// TIA Portal project "Module1.2" (V16)

(* hardware
DEVICE "S7-1200 station_1"  S7-1200 Station
   slot 0: "Rack_0"  S7-1200 Rack  Rack  V1.0
   slot 1: "PLC_1"  CPU 1214C DC/DC/DC  6ES7 214-1AG40-0XB0  V4.2
   slot 2: "DI 8/DQ 8x24VDC_1"  SM 1223 DI8/DQ8 x 24VDC  6ES7 223-1BH30-0XB0  V1.0
*)

// ===== PLC "PLC_1"  CPU 1214C DC/DC/DC =====

VAR_GLOBAL   // PLC tag table "Default tag table"
   "R" AT %Q2.1 : Bool;
   "embryoQuality" AT %M10.0 : Bool;
   "initialStep" AT %M0.0 : Bool;
   "reset" AT %M0.1 : Bool;
   "start" AT %M0.2 : Bool;
   "startConveyor" AT %M0.3 : Bool;
   "pushEmbryo" AT %M0.4 : Bool;
   "waitEmbryo" AT %M0.5 : Bool;
   "stopConveyor" AT %M0.6 : Bool;
   "grapEmbryo" AT %M0.7 : Bool;
   "goingUp" AT %M1.0 : Bool;
   "goingDown" AT %M1.1 : Bool;
   "goingRight" AT %M1.2 : Bool;
   "putEmbryoDown" AT %M1.3 : Bool;
   "checkEmbryo" AT %M1.4 : Bool;
   "realizeEmbryo" AT %M1.5 : Bool;
   "offSuction" AT %M1.6 : Bool;
   "fs" AT %I1.0 : Bool;
END_VAR

VAR_GLOBAL   // PLC tag table "Default tag table_1"
   "System_Byte" AT %MB100 : Byte;
   "FirstScan" AT %M100.0 : Bool;
   "DiagStatusUpdate" AT %M100.1 : Bool;
   "AlwaysTRUE" AT %M100.2 : Bool;
   "AlwaysFALSE" AT %M100.3 : Bool;
   "Clock_Byte" AT %MB200 : Byte;
   "Clock_10Hz" AT %M200.0 : Bool;
   "Clock_5Hz" AT %M200.1 : Bool;
   "Clock_2.5Hz" AT %M200.2 : Bool;
   "Clock_2Hz" AT %M200.3 : Bool;
   "Clock_1.25Hz" AT %M200.4 : Bool;
   "Clock_1Hz" AT %M200.5 : Bool;
   "Clock_0.625Hz" AT %M200.6 : Bool;
   "Clock_0.5Hz" AT %M200.7 : Bool;
   "startBTN" AT %I0.0 : Bool;
   "stopBTN" AT %I0.1 : Bool;
   "resetBTN" AT %I0.2 : Bool;
   "headConveyorSS" AT %I0.3 : Bool;
   "enConveyorSS" AT %I0.6 : Bool;
   "embryoSS" AT %I2.1 : Bool;
   "pushCompressLimit" AT %I0.7 : Bool;
   "pushExpandLimit" AT %I2.0 : Bool;
   "leftLimit" AT %I2.6 : Bool;
   "rightLimit" AT %I2.4 : Bool;
   "downLimit" AT %I2.2 : Bool;
   "upLimit" AT %I2.3 : Bool;
   "stopperCompressLimit" AT %I0.4 : Bool;
   "stopperExpandLimit" AT %I0.5 : Bool;
   "middleHCylinder" AT %I2.5 : Bool;
   "Push" AT %Q0.5 : Bool;
   "Left" AT %Q1.1 : Bool;
   "Right" AT %Q0.2 : Bool;
   "Down" AT %Q0.3 : Bool;
   "stopperDown" AT %Q0.0 : Bool;
   "Conveyor" AT %Q2.0 : Bool;
   "Suction" AT %Q0.4 : Bool;
   "Y" AT %Q2.3 : Bool;
   "G" AT %Q2.2 : Bool;
   "CBPL" AT %I2.7 : Bool;
END_VAR

// folder: System blocks/Program resources

DATA_BLOCK "timer1"   // DB1
{ S7_Optimized_Access := 'TRUE' }
AUTHOR : Simatic
FAMILY : IEC
NAME : IEC_TMR
VERSION : 1.0
// stored: InstanceOfName IEC_TIMER
"IEC_TIMER"
BEGIN
END_DATA_BLOCK

DATA_BLOCK "timer2"   // DB2
{ S7_Optimized_Access := 'TRUE' }
AUTHOR : Simatic
FAMILY : IEC
NAME : IEC_TMR
VERSION : 1.0
// stored: InstanceOfName IEC_TIMER
"IEC_TIMER"
BEGIN
END_DATA_BLOCK

DATA_BLOCK "timer3"   // DB3
{ S7_Optimized_Access := 'TRUE' }
AUTHOR : Simatic
FAMILY : IEC
NAME : IEC_TMR
VERSION : 1.0
// stored: InstanceOfName IEC_TIMER
"IEC_TIMER"
BEGIN
END_DATA_BLOCK

// folder: (top level)

ORGANIZATION_BLOCK "Main"   // OB1, LAD, ProgramCycle
TITLE = "Main Program Sweep (Cycle)"
{ S7_Optimized_Access := 'TRUE' }
VERSION : 0.1
   VAR_INPUT
      Initial_Call : Bool;   // Initial call of this OB
      Remanence : Bool;   // =True, if remanent data are available
   END_VAR
BEGIN

REGION Network 1
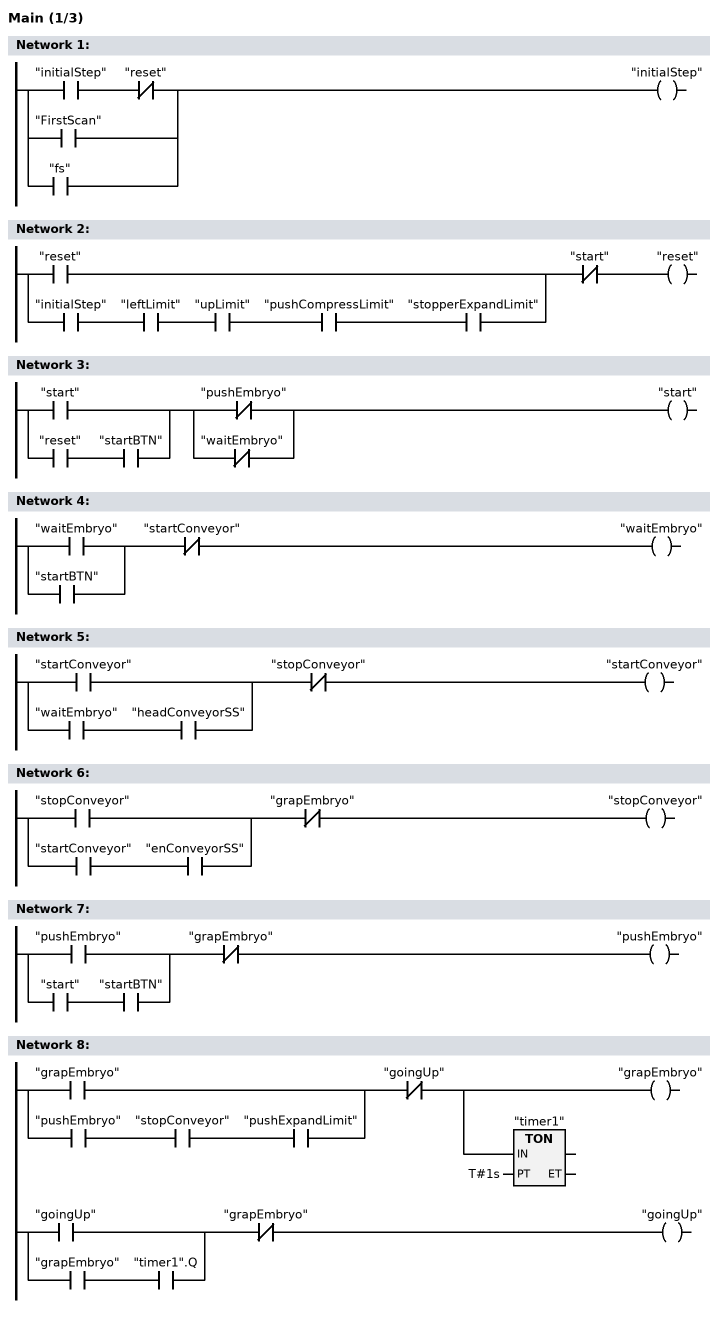
   RUNG wire#powerrail
      Contact( "initialStep" )
      I_Contact( "reset" )
      wire#w1
      Coil( "initialStep" )
   END_RUNG
   RUNG wire#powerrail
      Contact( "FirstScan" )
   END_RUNG wire#w1
   RUNG wire#powerrail
      Contact( "fs" )
   END_RUNG wire#w1
   // the same network as SCL:
   "initialStep" := ("initialStep" AND NOT "reset") OR "FirstScan" OR "fs";
END_REGION

REGION Network 2
   RUNG wire#powerrail
      Contact( "reset" )
      wire#w1
      I_Contact( "start" )
      Coil( "reset" )
   END_RUNG
   RUNG wire#powerrail
      Contact( "initialStep" )
      Contact( "leftLimit" )
      Contact( "upLimit" )
      Contact( "pushCompressLimit" )
      Contact( "stopperExpandLimit" )
   END_RUNG wire#w1
   // the same network as SCL:
   "reset" := ("reset" OR ("initialStep" AND "leftLimit" AND "upLimit" AND "pushCompressLimit" AND "stopperExpandLimit")) AND NOT "start";
END_REGION

REGION Network 3
   RUNG wire#powerrail
      Contact( "start" )
      wire#w1
      I_Contact( "pushEmbryo" )
      wire#w2
      Coil( "start" )
   END_RUNG
   RUNG wire#powerrail
      Contact( "reset" )
      Contact( "startBTN" )
   END_RUNG wire#w1
   RUNG wire#w1
      I_Contact( "waitEmbryo" )
   END_RUNG wire#w2
   // the same network as SCL:
   "start" := ("start" OR ("reset" AND "startBTN")) AND (NOT "pushEmbryo" OR NOT "waitEmbryo");
END_REGION

REGION Network 4
   RUNG wire#powerrail
      Contact( "waitEmbryo" )
      wire#w1
      I_Contact( "startConveyor" )
      Coil( "waitEmbryo" )
   END_RUNG
   RUNG wire#powerrail
      Contact( "startBTN" )
   END_RUNG wire#w1
   // the same network as SCL:
   "waitEmbryo" := ("waitEmbryo" OR "startBTN") AND NOT "startConveyor";
END_REGION

REGION Network 5
   RUNG wire#powerrail
      Contact( "startConveyor" )
      wire#w1
      I_Contact( "stopConveyor" )
      Coil( "startConveyor" )
   END_RUNG
   RUNG wire#powerrail
      Contact( "waitEmbryo" )
      Contact( "headConveyorSS" )
   END_RUNG wire#w1
   // the same network as SCL:
   "startConveyor" := ("startConveyor" OR ("waitEmbryo" AND "headConveyorSS")) AND NOT "stopConveyor";
END_REGION

REGION Network 6
   RUNG wire#powerrail
      Contact( "stopConveyor" )
      wire#w1
      I_Contact( "grapEmbryo" )
      Coil( "stopConveyor" )
   END_RUNG
   RUNG wire#powerrail
      Contact( "startConveyor" )
      Contact( "enConveyorSS" )
   END_RUNG wire#w1
   // the same network as SCL:
   "stopConveyor" := ("stopConveyor" OR ("startConveyor" AND "enConveyorSS")) AND NOT "grapEmbryo";
END_REGION

REGION Network 7
   RUNG wire#powerrail
      Contact( "pushEmbryo" )
      wire#w1
      I_Contact( "grapEmbryo" )
      Coil( "pushEmbryo" )
   END_RUNG
   RUNG wire#powerrail
      Contact( "start" )
      Contact( "startBTN" )
   END_RUNG wire#w1
   // the same network as SCL:
   "pushEmbryo" := ("pushEmbryo" OR ("start" AND "startBTN")) AND NOT "grapEmbryo";
END_REGION

REGION Network 8
   "grapEmbryo" := ("grapEmbryo" OR ("pushEmbryo" AND "stopConveyor" AND "pushExpandLimit")) AND NOT "goingUp";
   "timer1".TON(IN := "grapEmbryo", PT := T#1s);
   "goingUp" := ("goingUp" OR ("grapEmbryo" AND "timer1".Q)) AND NOT "grapEmbryo";
END_REGION

REGION Network 9
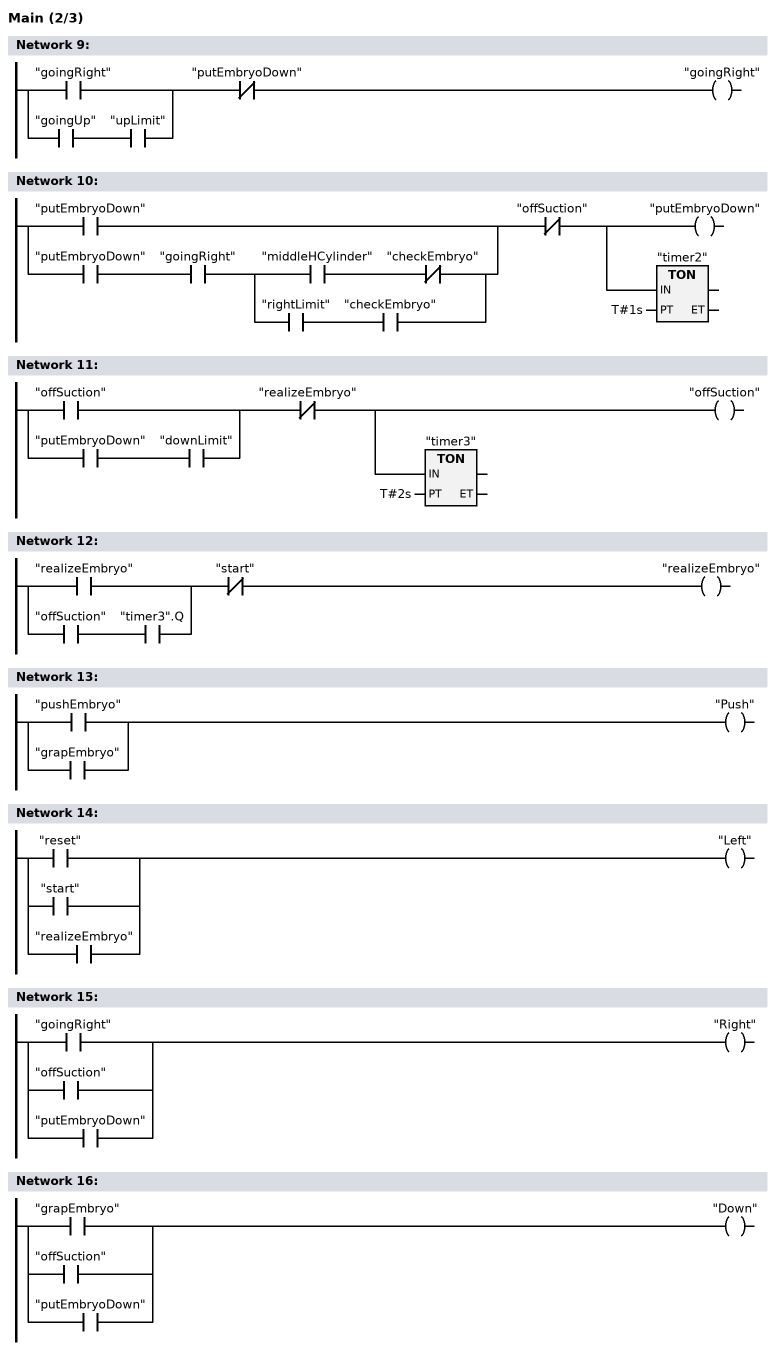
   RUNG wire#powerrail
      Contact( "goingRight" )
      wire#w1
      I_Contact( "putEmbryoDown" )
      Coil( "goingRight" )
   END_RUNG
   RUNG wire#powerrail
      Contact( "goingUp" )
      Contact( "upLimit" )
   END_RUNG wire#w1
   // the same network as SCL:
   "goingRight" := ("goingRight" OR ("goingUp" AND "upLimit")) AND NOT "putEmbryoDown";
END_REGION

REGION Network 10
   "putEmbryoDown" := ("putEmbryoDown" OR ("putEmbryoDown" AND "goingRight" AND (("middleHCylinder" AND NOT "checkEmbryo") OR ("rightLimit" AND "checkEmbryo")))) AND NOT "offSuction";
   "timer2".TON(IN := "putEmbryoDown", PT := T#1s);
END_REGION

REGION Network 11
   "offSuction" := ("offSuction" OR ("putEmbryoDown" AND "downLimit")) AND NOT "realizeEmbryo";
   "timer3".TON(IN := "offSuction", PT := T#2s);
END_REGION

REGION Network 12
   RUNG wire#powerrail
      Contact( "realizeEmbryo" )
      wire#w1
      I_Contact( "start" )
      Coil( "realizeEmbryo" )
   END_RUNG
   RUNG wire#powerrail
      Contact( "offSuction" )
      Contact( "timer3".Q )
   END_RUNG wire#w1
   // the same network as SCL:
   "realizeEmbryo" := ("realizeEmbryo" OR ("offSuction" AND "timer3".Q)) AND NOT "start";
END_REGION

REGION Network 13
   RUNG wire#powerrail
      Contact( "pushEmbryo" )
      wire#w1
      Coil( "Push" )
   END_RUNG
   RUNG wire#powerrail
      Contact( "grapEmbryo" )
   END_RUNG wire#w1
   // the same network as SCL:
   "Push" := "pushEmbryo" OR "grapEmbryo";
END_REGION

REGION Network 14
   RUNG wire#powerrail
      Contact( "reset" )
      wire#w1
      Coil( "Left" )
   END_RUNG
   RUNG wire#powerrail
      Contact( "start" )
   END_RUNG wire#w1
   RUNG wire#powerrail
      Contact( "realizeEmbryo" )
   END_RUNG wire#w1
   // the same network as SCL:
   "Left" := "reset" OR "start" OR "realizeEmbryo";
END_REGION

REGION Network 15
   RUNG wire#powerrail
      Contact( "goingRight" )
      wire#w1
      Coil( "Right" )
   END_RUNG
   RUNG wire#powerrail
      Contact( "offSuction" )
   END_RUNG wire#w1
   RUNG wire#powerrail
      Contact( "putEmbryoDown" )
   END_RUNG wire#w1
   // the same network as SCL:
   "Right" := "goingRight" OR "offSuction" OR "putEmbryoDown";
END_REGION

REGION Network 16
   RUNG wire#powerrail
      Contact( "grapEmbryo" )
      wire#w1
      Coil( "Down" )
   END_RUNG
   RUNG wire#powerrail
      Contact( "offSuction" )
   END_RUNG wire#w1
   RUNG wire#powerrail
      Contact( "putEmbryoDown" )
   END_RUNG wire#w1
   // the same network as SCL:
   "Down" := "grapEmbryo" OR "offSuction" OR "putEmbryoDown";
END_REGION

REGION Network 17
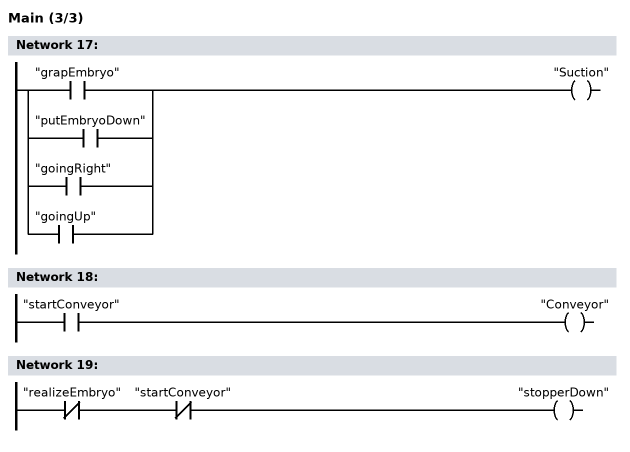
   RUNG wire#powerrail
      Contact( "grapEmbryo" )
      wire#w1
      Coil( "Suction" )
   END_RUNG
   RUNG wire#powerrail
      Contact( "putEmbryoDown" )
   END_RUNG wire#w1
   RUNG wire#powerrail
      Contact( "goingRight" )
   END_RUNG wire#w1
   RUNG wire#powerrail
      Contact( "goingUp" )
   END_RUNG wire#w1
   // the same network as SCL:
   "Suction" := "grapEmbryo" OR "putEmbryoDown" OR "goingRight" OR "goingUp";
END_REGION

REGION Network 18
   RUNG wire#powerrail
      Contact( "startConveyor" )
      Coil( "Conveyor" )
   END_RUNG
   // the same network as SCL:
   "Conveyor" := "startConveyor";
END_REGION

REGION Network 19
   RUNG wire#powerrail
      I_Contact( "realizeEmbryo" )
      I_Contact( "startConveyor" )
      Coil( "stopperDown" )
   END_RUNG
   // the same network as SCL:
   "stopperDown" := NOT "realizeEmbryo" AND NOT "startConveyor";
END_REGION
END_ORGANIZATION_BLOCK